PROGRAM PRG_ZeroOrder_PMPS
VAR
// PMPS
    ffZeroOrderBeam : FB_FastFault := (
        i_xAutoReset := TRUE,
        i_DevName := 'Zero Order Beam',
        i_Desc := 'Faults when Zero order beam safe conditions are not met',
        i_TypeCode := 16#F506);
    {attribute 'pytmc' := '
        pv: @(PREFIX)SafeBenderRange
        field: ZNAM FALSE
        field: ONAM TRUE
    '}
    bSafeBenderRange : BOOL;

    {attribute 'pytmc' := '
        pv: @(PREFIX)LRG_Grating_IN
        field: ZNAM FALSE
        field: ONAM TRUE
    '}
    bLRG_Grating_IN : BOOL;

    {attribute 'pytmc' := '
        pv: @(PREFIX)MEG_Grating_IN
        field: ZNAM FALSE
        field: ONAM TRUE
    '}
    bMEG_Grating_IN : BOOL;

    {attribute 'pytmc' := '
        pv: @(PREFIX)HEG_Grating_IN
        field: ZNAM FALSE
        field: ONAM TRUE
    '}
    bHEG_Grating_IN : BOOL;

    {attribute 'pytmc' := '
        pv: @(PREFIX)LEG_Grating_IN
        field: ZNAM FALSE
        field: ONAM TRUE
    '}
    bLEG_Grating_IN : BOOL;

    {attribute 'pytmc' := '
        pv: @(PREFIX)ZOS_IN
        field: ZNAM FALSE
        field: ONAM TRUE
    '}
    bZOS_IN : BOOL;

    {attribute 'pytmc' := '
        pv: @(PREFIX)ZOB_on_Lower_Stopper
        field: ZNAM FALSE
        field: ONAM TRUE
    '}
    bZOB_on_Lower_Stopper : BOOL;

    {attribute 'pytmc' := '
        pv: @(PREFIX)MR1K1_Inserted
        field: ZNAM FALSE
        field: ONAM TRUE
    '}
    bMR1K1_Inserted : BOOL;



    {attribute 'pytmc' := '
        pv: @(PREFIX)MachineMode
        field: ZRST NC
        field: ONST SC
        field: TWST Misconfig
        field: THST UnInit
    '}
    nMachineMode : INT;

    {attribute 'pytmc' := '
        pv: @(PREFIX)BeamPermitted
        field: ZNAM FALSE
        field: ONAM TRUE
    '}
    bBeamPermitted : BOOL;


    Pm3 : LREAL;
    Pm2: LREAL;
    Pm1: LREAL;
    Hm1: LREAL;
    HZos:LREAL;
    Zbm1: LREAL;
    Zbm2: LREAL;
    Zbm3: LREAL;
    Hbm1: LREAL;
    Hbm2: LREAL;
    Hbm3: LREAL;
    Hb0m3:LREAL;
    //fixed calc
    Hm3	 : LREAL;
    Hpiv : LREAL;
    Theta_m1: LREAL;
    Theta_m2: LREAL;
    Theta_m3: LREAL;
    {attribute 'pytmc' := '
        pv: @(PREFIX)Delta
        field: ZNAM FALSE
        field: ONAM TRUE
    '}
    Delta : LREAL;
    Ans : LREAL;
    ffZeroOrderBeamExitSlits : FB_FastFault := (
        i_xAutoReset := TRUE,
        i_DevName := 'Zero Order Beam and Exit Slits',
        i_Desc := 'Faults when Zero order beam is aligned and exit slits are closed',
        i_TypeCode := 16#F506);
    mm: INT;
    eV: INT;
END_VAR
VAR CONSTANT
    Hi2 :LREAL:=1.4;//m
    Zi2: LREAL :=731.613;//m
    Theta0 : LREAL:=0;
    Zm1 : LREAL:=733.772;//m
    Zmon : LREAL:=739.622;//m
    Zpiv : LREAL:= 739.762 ; //m
    Zzos : LREAL:= 741.422;//m
    Pm1Offset: LREAL:= 18081.1;
    Pm2Offset: LREAL:= -90603;
    Pm3Offset: LREAL:= -63300;//urad, could depend on the inserted grating
END_VAR


//Diagnostics
bSafeBenderRange := SafeBenderRange();
nMachineMode := PMPS_GVL.stCurrentBeamParameters.nMachineMode;
bMR1K1_Inserted := MR1K1_Inserted();
ACT_Grating_IN();
ACT_CALC();
ACT_ZOS_IN();
ACT_ExitSlitsGap();

//Is the ZO beam on the stopper? TRUE if Hzos - hb0m3(Zzoz)  > Δ
(*
    Δ=2.0 mm for LRG @ >1000 eV
    Δ=2.5 mm for LRG @ <1000 eV
    Δ=3.0 mm for LRG @ <550 eV
    Δ=6.0 mm for LEG, MEG, HEG
*)
Ans := (Hzos*1E3) - Hb0m3; //um

IF bLRG_Grating_IN AND GVL_PMPS.rPhotonEnergy <550 THEN Delta := 3*1E3(*um*);
ELSIF bLRG_Grating_IN AND GVL_PMPS.rPhotonEnergy <1000 THEN Delta := 2.5*1E3(*um*);
ELSIF bLRG_Grating_IN AND GVL_PMPS.rPhotonEnergy >=1000 THEN Delta := 2*1E3(*um*);
ELSIF (bMEG_Grating_IN OR bHEG_Grating_IN OR bLEG_Grating_IN) THEN Delta := 6*1E3(*um*);
ELSE	Delta := Ans;
END_IF

bZOB_on_Lower_Stopper := Ans > Delta;


ffZeroOrderBeam.i_xOK := (SafeBenderRange() AND (((PMPS_GVL.stCurrentBeamParameters.nMachineMode =1(*SC*)) AND (PMPS_GVL.stCurrentBeamParameters.nBeamClass <=6)) OR (PMPS_GVL.stCurrentBeamParameters.nMachineMode =0(*NC*))))
                OR (bLRG_Grating_IN AND bZOS_IN AND bZOB_on_Lower_Stopper AND MR1K1_Inserted()(*NC or SC Any Beamclass with beam at ZOS*))
                OR ((bMEG_Grating_IN OR bHEG_Grating_IN OR bLEG_Grating_IN) AND bZOS_IN AND bZOB_on_Lower_Stopper AND MR1K1_Inserted()(*NC or SC Any Beamclass with beam at ZOS*));
ffZeroOrderBeam(io_fbFFHWO := GVL_PMPS.fbFastFaultOutput1);
bBeamPermitted := ffZeroOrderBeam.i_xOK;

//

ACTION ACT_CALC:
///calc
//Hm1 = 1400000+mr1k1 ben Y up
Hm1:= 1400000+M12.stAxisStatus.fActPosition; //um
//Pm1 = Pm1Offset + mr1k1 bend pitch
Pm1 := Pm1Offset + Main.M16.stAxisStatus.fActPosition; //urad
//Hpiv = 1.625427 is correction from nominal
Hpiv:= (1.625247)*1E6; //um
//Pm2 = mono mirror pitch + Pm2Offset urad
Pm2 := Main.M6.stAxisStatus.fActPosition + Pm2Offset;//urad
//Hm3 = Hpiv + 0.006 m
Hm3:= Hpiv + (0.006*1E6); //um
//Pm3 = mono grating pitch + Pm3Offset urad
Pm3 := Main.M7.stAxisStatus.fActPosition + Pm3Offset; //urad
//Hzos = 1824.3 + st1k1_zos mm
Hzos:= 1824.3 + M24.stAxisStatus.fActPosition; //mm


//urad
Theta_m1 := 2*Pm1 - Theta0;
Theta_m2 := 2*Pm2 - Theta_m1;
Theta_m3 := 2 *Pm3 - 2 * Pm2 + 2* Pm1 - Theta0;

// fix units
//um
Zbm1 := (Hm1 - TAN(Pm1*1E-6)* (Zm1*1E6) - (Hi2*1E6) + TAN(Theta0*1E-6) *(Zi2*1E6))/(TAN(Theta0*1E-6) - TAN(Pm1*1E-6));
hbm1 := TAN(Pm1*1E-6)*Zbm1 + Hm1 - TAN(Pm1*1E-6)*(Zm1*1E6);
//u?
Zbm2 := (Hbm1 - TAN(Theta_m1*1E-6)*Zbm1 - Hpiv + TAN(Pm2*1E-6)*(Zpiv*1E6))/ (TAN(Pm2*1E-6) - TAN(Theta_m1*1E-6));
Hbm2 := TAN(Pm2*1E-6)*Zbm2 + Hpiv - TAN(Pm2*1E-6)*(Zpiv*1E6);

Zbm3 := (Hbm2 - TAN(Theta_m2*1E-6)*Zbm2 - Hm3 + TAN(Pm3*1E-6)*(Zpiv*1E6))/ (TAN(Pm3*1E-6) - TAN(Theta_m2*1E-6));
Hbm3 := TAN(Pm3*1E-6) * Zbm3 + Hm3 - TAN(Pm3*1E-6)*(Zpiv*1E6);

Hb0m3 := TAN(Theta_m3*1E-6)*(Zzos*1E6) + Hbm3 - TAN(Theta_m3*1E-6)*Zbm3;
END_ACTION

ACTION ACT_ExitSlitsGap:
// FAULT condition: Hzos -1.0mm <= Hb0m3) AND sl1k2 gap <= 8.0 mm
ffZeroOrderBeamExitSlits.i_xOK := NOT( (( (Hzos*1E3) - 1) <= Hb0m3) AND ( M22.stAxisStatus.fActPosition <= 8000(*um*)));
ffZeroOrderBeamExitSlits(io_fbFFHWO := GVL_PMPS.fbFastFaultOutput1);
END_ACTION

ACTION ACT_Grating_IN:
bLRG_Grating_IN := PRG_SP1K1_MONO.eStateGet = E_Grating_States.LRG;
bMEG_Grating_IN := PRG_SP1K1_MONO.eStateGet = E_Grating_States.MEG;
bHEG_Grating_IN := PRG_SP1K1_MONO.eStateGet = E_Grating_States.HEG;
bLEG_Grating_IN := PRG_SP1K1_MONO.eStateGet = E_Grating_States.LEG;
END_ACTION

ACTION ACT_ZOS_IN:
IF GVL_PMPS.rPhotonEnergy >1500 THEN bZOS_IN:= FALSE;
    ELSIF (GVL_PMPS.rPhotonEnergy >1000 AND M24.stAxisStatus.fActPosition>= 8.5) THEN bZOS_IN:= TRUE;
        ELSIF (GVL_PMPS.rPhotonEnergy <=1000 AND GVL_PMPS.rPhotonEnergy >550 AND M24.stAxisStatus.fActPosition>= 7.9) THEN bZOS_IN:= TRUE;
            ELSIF (GVL_PMPS.rPhotonEnergy <=550 AND GVL_PMPS.rPhotonEnergy >200 AND M24.stAxisStatus.fActPosition>= 6.9) THEN bZOS_IN:= TRUE;
                ELSE bZOS_IN:= FALSE;
END_IF
END_ACTION

METHOD MR1K1_Inserted : BOOL
VAR_INPUT
END_VAR
MR1K1_Inserted := PMPS_GVL.stCurrentBeamParameters.aVetoDevices[PMPS.K_Stopper.MR1K1_IN]
                    AND NOT PMPS_GVL.stCurrentBeamParameters.aVetoDevices[PMPS.K_Stopper.MR1K1_OUT];
END_METHOD

METHOD SafeBenderRange : BOOL
VAR_INPUT
END_VAR
 SafeBenderRange :=  GVL_M1K1_BENDER_Constants.nM1K1bendUS_PMPS_LowerLimit < M17.nEncoderCount AND M17.nEncoderCount < GVL_M1K1_BENDER_Constants.nM1K1bendUS_PMPS_UpperLimit AND
    GVL_M1K1_BENDER_Constants.nM1K1bendDS_PMPS_LowerLimit < M18.nEncoderCount AND M18.nEncoderCount < GVL_M1K1_BENDER_Constants.nM1K1bendDS_PMPS_UpperLimit;
END_METHOD

END_PROGRAM

(* stored: Version 1.1.0.1, ProductVersion 3.1.4024.12
   POU PRG_ZeroOrder_PMPS: Id {91b5156c-1864-44ab-9bf4-9660205ee3fe}, SpecialFunc None
   Action ACT_CALC: Id {29570aa5-9d14-46b0-b59e-651abe0f5e16}
   Action ACT_ExitSlitsGap: Id {72615217-f71d-41ee-b0dd-e3c54f411832}
   Action ACT_Grating_IN: Id {def557f5-6fcd-48fa-9e2d-d3f3ab8c4d09}
   Action ACT_ZOS_IN: Id {ea635b1c-413a-4430-b9a8-7a35a57ab8c1}
   Method MR1K1_Inserted: Id {a6f63631-54cf-4bad-bff6-69bbc818c904}
   Method SafeBenderRange: Id {b4c0e9bb-a0bf-4708-9d0f-639acbeed916} *)
